FUNCTION_BLOCK FB_Module01 EXTENDS FB_Module
VAR_INPUT
END_VAR
VAR_OUTPUT
END_VAR
VAR
	fbComponent0:				FB_ComponentEx;
	fbComponent1:				FB_ComponentEx;
	fbComponent2:				FB_ComponentEx;
END_VAR

// https://peterzerlauth.com/
SUPER^();

bHomed S= bHomePosition;

fbComponent0();
fbComponent1();
fbComponent2();

METHOD PROTECTED M_Execute : bool
VAR_INPUT
END_VAR
VAR
	bReturn:					BOOL:= TRUE;
END_VAR
CASE fbSequence.P_Number OF
	E_Sequence.Start:
		bReturn:= TRUE;
		fbSequence.M_Await('Start 0', T#0S , T#1S, TRUE, bReturn, 10);
	
	10:
		bReturn:= TRUE;
		fbSequence.M_Await('Step 10', T#0S, T#0S, TRUE, bReturn, 20);
		
	20:
		bReturn:= FALSE;
		fbSequence.M_Await('Step 20', T#1S, T#0S, FALSE, bReturn, E_Sequence.Done);	
		
	E_Sequence.Done:
		fbSequence.M_Reset();

END_CASE

// IF bWarning THEN
// 	fbEvent.M_Warning('My secound Warning', 19 );	
// END_IF
END_METHOD

METHOD PROTECTED M_Initialise : BOOL
VAR_INPUT
END_VAR
M_Initialise:= SUPER^.M_Initialise();

P_Info.P_ID:= 'M001';

fbMembers.M_Attach(THIS^, fbComponent0);
fbMembers.M_Attach(THIS^, fbComponent1);
fbMembers.M_Attach(THIS^, fbComponent2);
END_METHOD

METHOD PROTECTED M_Running
VAR_INPUT
END_VAR
IF NOT IO.bOn THEN
	fbEvent.M_AddSTRING('BMK1');
	fbEvent.M_Abort('Power not on  %s', 15);
ELSIF NOT IO.bEMStop THEN
	fbEvent.M_AddSTRING('BMK2');
	fbEvent.M_Abort('Emergency stop not ok %s', 16);
ELSIF NOT IO.bDoorsOk THEN
	fbEvent.M_AddSTRING('BMK3');
	fbEvent.M_Stop('Door Not OK', 17);	
ELSIF NOT IO.bFuse THEN	
	fbEvent.M_Stop('Fuse Triped', 18);		
END_IF
END_METHOD

METHOD PROTECTED M_Starting : BOOL
VAR_INPUT
END_VAR
M_Starting:= SUPER^.M_Starting();
END_METHOD

METHOD PROTECTED M_Stopping : BOOL // Return state complete
VAR_INPUT
END_VAR
// State Stopping
M_Stopping:= SUPER^.M_Stopping();
END_METHOD

END_FUNCTION_BLOCK

(* stored: Version 1.1.0.1
   POU FB_Module01: Id {3744d03d-359c-4ab8-84fb-4ea93b7a5162}, SpecialFunc None
   Method M_Execute: Id {0f7f4331-8af5-0744-015a-f65d0021dd06}
   Method M_Initialise: Id {714c485c-83a6-4af2-a706-fec3f6b598e5}
   Method M_Running: Id {eaffebca-5ff2-4f17-be84-3310a9ace22e}
   Method M_Starting: Id {6f002794-61fc-043c-1d84-a8bc502c5d3a}
   Method M_Stopping: Id {478c517c-d184-0eaf-2697-597088f6cf3f} *)
